	counter9337: LREAL :=  0;
	counter9338: LREAL :=  0;
	counter9339: LREAL :=  0;
	counter9340: LREAL :=  0;
	counter9341: LREAL :=  0;
	counter9342: LREAL :=  0;
	counter9343: LREAL :=  0;
	counter9344: LREAL :=  0;
	counter9345: LREAL :=  0;
	counter9346: LREAL :=  0;
	counter9347: LREAL :=  0;
	counter9348: LREAL :=  0;
	counter9349: LREAL :=  0;
	counter9350: LREAL :=  0;
	counter9351: LREAL :=  0;
	counter9352: LREAL :=  0;
	counter9353: LREAL :=  0;
	counter9354: LREAL :=  0;
	counter9355: LREAL :=  0;
	counter9356: LREAL :=  0;
	counter9357: LREAL :=  0;
	counter9358: LREAL :=  0;
	counter9359: LREAL :=  0;
	counter9360: LREAL :=  0;
	counter9361: LREAL :=  0;
	counter9362: LREAL :=  0;
	counter9363: LREAL :=  0;
	counter9364: LREAL :=  0;
	counter9365: LREAL :=  0;
	counter9366: LREAL :=  0;
	counter9367: LREAL :=  0;
	counter9368: LREAL :=  0;
	counter9369: LREAL :=  0;
	counter9370: LREAL :=  0;
	counter9371: LREAL :=  0;
	counter9372: LREAL :=  0;
	counter9373: LREAL :=  0;
	counter9374: LREAL :=  0;
	counter9375: LREAL :=  0;
	counter9376: LREAL :=  0;
	counter9377: LREAL :=  0;
	counter9378: LREAL :=  0;
	counter9379: LREAL :=  0;
	counter9380: LREAL :=  0;
	counter9381: LREAL :=  0;
	counter9382: LREAL :=  0;
	counter9383: LREAL :=  0;
	counter9384: LREAL :=  0;
	counter9385: LREAL :=  0;
	counter9386: LREAL :=  0;
	counter9387: LREAL :=  0;
	counter9388: LREAL :=  0;
	counter9389: LREAL :=  0;
	counter9390: LREAL :=  0;
	counter9391: LREAL :=  0;
	counter9392: LREAL :=  0;
	counter9393: LREAL :=  0;
	counter9394: LREAL :=  0;
	counter9395: LREAL :=  0;
	counter9396: LREAL :=  0;
	counter9397: LREAL :=  0;
	counter9398: LREAL :=  0;
	counter9399: LREAL :=  0;
	counter9400: LREAL :=  0;
	counter9401: LREAL :=  0;
	counter9402: LREAL :=  0;
	counter9403: LREAL :=  0;
	counter9404: LREAL :=  0;
	counter9405: LREAL :=  0;
	counter9406: LREAL :=  0;
	counter9407: LREAL :=  0;
	counter9408: LREAL :=  0;
	counter9409: LREAL :=  0;
	counter9410: LREAL :=  0;
	counter9411: LREAL :=  0;
	counter9412: LREAL :=  0;
	counter9413: LREAL :=  0;
	counter9414: LREAL :=  0;
	counter9415: LREAL :=  0;
	counter9416: LREAL :=  0;
	counter9417: LREAL :=  0;
	counter9418: LREAL :=  0;
	counter9419: LREAL :=  0;
	counter9420: LREAL :=  0;
	counter9421: LREAL :=  0;
	counter9422: LREAL :=  0;
	counter9423: LREAL :=  0;
	counter9424: LREAL :=  0;
	counter9425: LREAL :=  0;
	counter9426: LREAL :=  0;
	counter9427: LREAL :=  0;
	counter9428: LREAL :=  0;
	counter9429: LREAL :=  0;
	counter9430: LREAL :=  0;
	counter9431: LREAL :=  0;
	counter9432: LREAL :=  0;
	counter9433: LREAL :=  0;
	counter9434: LREAL :=  0;
	counter9435: LREAL :=  0;
	counter9436: LREAL :=  0;
	counter9437: LREAL :=  0;
	counter9438: LREAL :=  0;
	counter9439: LREAL :=  0;
	counter9440: LREAL :=  0;
	counter9441: LREAL :=  0;
	counter9442: LREAL :=  0;
	counter9443: LREAL :=  0;
	counter9444: LREAL :=  0;
	counter9445: LREAL :=  0;
	counter9446: LREAL :=  0;
	counter9447: LREAL :=  0;
	counter9448: LREAL :=  0;
	counter9449: LREAL :=  0;
	counter9450: LREAL :=  0;
	counter9451: LREAL :=  0;
	counter9452: LREAL :=  0;
	counter9453: LREAL :=  0;
	counter9454: LREAL :=  0;
	counter9455: LREAL :=  0;
	counter9456: LREAL :=  0;
	counter9457: LREAL :=  0;
	counter9458: LREAL :=  0;
	counter9459: LREAL :=  0;
	counter9460: LREAL :=  0;
	counter9461: LREAL :=  0;
	counter9462: LREAL :=  0;
	counter9463: LREAL :=  0;
	counter9464: LREAL :=  0;
	counter9465: LREAL :=  0;
	counter9466: LREAL :=  0;
	counter9467: LREAL :=  0;
	counter9468: LREAL :=  0;
	counter9469: LREAL :=  0;
	counter9470: LREAL :=  0;
	counter9471: LREAL :=  0;
	counter9472: LREAL :=  0;
	counter9473: LREAL :=  0;
	counter9474: LREAL :=  0;
	counter9475: LREAL :=  0;
	counter9476: LREAL :=  0;
	counter9477: LREAL :=  0;
	counter9478: LREAL :=  0;
	counter9479: LREAL :=  0;
	counter9480: LREAL :=  0;
	counter9481: LREAL :=  0;
	counter9482: LREAL :=  0;
	counter9483: LREAL :=  0;
	counter9484: LREAL :=  0;
	counter9485: LREAL :=  0;
	counter9486: LREAL :=  0;
	counter9487: LREAL :=  0;
	counter9488: LREAL :=  0;
	counter9489: LREAL :=  0;
	counter9490: LREAL :=  0;
	counter9491: LREAL :=  0;
	counter9492: LREAL :=  0;
	counter9493: LREAL :=  0;
	counter9494: LREAL :=  0;
	counter9495: LREAL :=  0;
	counter9496: LREAL :=  0;
	counter9497: LREAL :=  0;
	counter9498: LREAL :=  0;
	counter9499: LREAL :=  0;
	counter9500: LREAL :=  0;
	counter9501: LREAL :=  0;
	counter9502: LREAL :=  0;
	counter9503: LREAL :=  0;
	counter9504: LREAL :=  0;
	counter9505: LREAL :=  0;
	counter9506: LREAL :=  0;
	counter9507: LREAL :=  0;
	counter9508: LREAL :=  0;
	counter9509: LREAL :=  0;
	counter9510: LREAL :=  0;
	counter9511: LREAL :=  0;
	counter9512: LREAL :=  0;
	counter9513: LREAL :=  0;
	counter9514: LREAL :=  0;
	counter9515: LREAL :=  0;
	counter9516: LREAL :=  0;
	counter9517: LREAL :=  0;
	counter9518: LREAL :=  0;
	counter9519: LREAL :=  0;
	counter9520: LREAL :=  0;
	counter9521: LREAL :=  0;
	counter9522: LREAL :=  0;
	counter9523: LREAL :=  0;
	counter9524: LREAL :=  0;
	counter9525: LREAL :=  0;
	counter9526: LREAL :=  0;
	counter9527: LREAL :=  0;
	counter9528: LREAL :=  0;
	counter9529: LREAL :=  0;
	counter9530: LREAL :=  0;
	counter9531: LREAL :=  0;
	counter9532: LREAL :=  0;
	counter9533: LREAL :=  0;
	counter9534: LREAL :=  0;
	counter9535: LREAL :=  0;
	counter9536: LREAL :=  0;
	counter9537: LREAL :=  0;
	counter9538: LREAL :=  0;
	counter9539: LREAL :=  0;
	counter9540: LREAL :=  0;
	counter9541: LREAL :=  0;
	counter9542: LREAL :=  0;
	counter9543: LREAL :=  0;
	counter9544: LREAL :=  0;
	counter9545: LREAL :=  0;
	counter9546: LREAL :=  0;
	counter9547: LREAL :=  0;
	counter9548: LREAL :=  0;
	counter9549: LREAL :=  0;
	counter9550: LREAL :=  0;
	counter9551: LREAL :=  0;
	counter9552: LREAL :=  0;
	counter9553: LREAL :=  0;
	counter9554: LREAL :=  0;
	counter9555: LREAL :=  0;
	counter9556: LREAL :=  0;
	counter9557: LREAL :=  0;
	counter9558: LREAL :=  0;
	counter9559: LREAL :=  0;
	counter9560: LREAL :=  0;
	counter9561: LREAL :=  0;
	counter9562: LREAL :=  0;
	counter9563: LREAL :=  0;
	counter9564: LREAL :=  0;
	counter9565: LREAL :=  0;
	counter9566: LREAL :=  0;
	counter9567: LREAL :=  0;
	counter9568: LREAL :=  0;
	counter9569: LREAL :=  0;
	counter9570: LREAL :=  0;
	counter9571: LREAL :=  0;
	counter9572: LREAL :=  0;
	counter9573: LREAL :=  0;
	counter9574: LREAL :=  0;
	counter9575: LREAL :=  0;
	counter9576: LREAL :=  0;
	counter9577: LREAL :=  0;
	counter9578: LREAL :=  0;
	counter9579: LREAL :=  0;
	counter9580: LREAL :=  0;
	counter9581: LREAL :=  0;
	counter9582: LREAL :=  0;
	counter9583: LREAL :=  0;
	counter9584: LREAL :=  0;
	counter9585: LREAL :=  0;
	counter9586: LREAL :=  0;
	counter9587: LREAL :=  0;
	counter9588: LREAL :=  0;
	counter9589: LREAL :=  0;
	counter9590: LREAL :=  0;
	counter9591: LREAL :=  0;
	counter9592: LREAL :=  0;
	counter9593: LREAL :=  0;
	counter9594: LREAL :=  0;
	counter9595: LREAL :=  0;
	counter9596: LREAL :=  0;
	counter9597: LREAL :=  0;
	counter9598: LREAL :=  0;
	counter9599: LREAL :=  0;
	counter9600: LREAL :=  0;
	counter9601: LREAL :=  0;
	counter9602: LREAL :=  0;
	counter9603: LREAL :=  0;
	counter9604: LREAL :=  0;
	counter9605: LREAL :=  0;
	counter9606: LREAL :=  0;
	counter9607: LREAL :=  0;
	counter9608: LREAL :=  0;
	counter9609: LREAL :=  0;
	counter9610: LREAL :=  0;
	counter9611: LREAL :=  0;
	counter9612: LREAL :=  0;
	counter9613: LREAL :=  0;
	counter9614: LREAL :=  0;
	counter9615: LREAL :=  0;
	counter9616: LREAL :=  0;
	counter9617: LREAL :=  0;
	counter9618: LREAL :=  0;
	counter9619: LREAL :=  0;
	counter9620: LREAL :=  0;
	counter9621: LREAL :=  0;
	counter9622: LREAL :=  0;
	counter9623: LREAL :=  0;
	counter9624: LREAL :=  0;
	counter9625: LREAL :=  0;
	counter9626: LREAL :=  0;
	counter9627: LREAL :=  0;
	counter9628: LREAL :=  0;
	counter9629: LREAL :=  0;
	counter9630: LREAL :=  0;
	counter9631: LREAL :=  0;
	counter9632: LREAL :=  0;
	counter9633: LREAL :=  0;
	counter9634: LREAL :=  0;
	counter9635: LREAL :=  0;
	counter9636: LREAL :=  0;
	counter9637: LREAL :=  0;
	counter9638: LREAL :=  0;
	counter9639: LREAL :=  0;
	counter9640: LREAL :=  0;
	counter9641: LREAL :=  0;
	counter9642: LREAL :=  0;
	counter9643: LREAL :=  0;
	counter9644: LREAL :=  0;
	counter9645: LREAL :=  0;
	counter9646: LREAL :=  0;
	counter9647: LREAL :=  0;
	counter9648: LREAL :=  0;
	counter9649: LREAL :=  0;
	counter9650: LREAL :=  0;
	counter9651: LREAL :=  0;
	counter9652: LREAL :=  0;
	counter9653: LREAL :=  0;
	counter9654: LREAL :=  0;
	counter9655: LREAL :=  0;
	counter9656: LREAL :=  0;
	counter9657: LREAL :=  0;
	counter9658: LREAL :=  0;
	counter9659: LREAL :=  0;
	counter9660: LREAL :=  0;
	counter9661: LREAL :=  0;
	counter9662: LREAL :=  0;
	counter9663: LREAL :=  0;
	counter9664: LREAL :=  0;
	counter9665: LREAL :=  0;
	counter9666: LREAL :=  0;
	counter9667: LREAL :=  0;
	counter9668: LREAL :=  0;
	counter9669: LREAL :=  0;
	counter9670: LREAL :=  0;
	counter9671: LREAL :=  0;
	counter9672: LREAL :=  0;
	counter9673: LREAL :=  0;
	counter9674: LREAL :=  0;
	counter9675: LREAL :=  0;
	counter9676: LREAL :=  0;
	counter9677: LREAL :=  0;
	counter9678: LREAL :=  0;
	counter9679: LREAL :=  0;
	counter9680: LREAL :=  0;
	counter9681: LREAL :=  0;
	counter9682: LREAL :=  0;
	counter9683: LREAL :=  0;
	counter9684: LREAL :=  0;
	counter9685: LREAL :=  0;
	counter9686: LREAL :=  0;
	counter9687: LREAL :=  0;
	counter9688: LREAL :=  0;
	counter9689: LREAL :=  0;
	counter9690: LREAL :=  0;
	counter9691: LREAL :=  0;
	counter9692: LREAL :=  0;
	counter9693: LREAL :=  0;
	counter9694: LREAL :=  0;
	counter9695: LREAL :=  0;
	counter9696: LREAL :=  0;
	counter9697: LREAL :=  0;
	counter9698: LREAL :=  0;
	counter9699: LREAL :=  0;
	counter9700: LREAL :=  0;
	counter9701: LREAL :=  0;
	counter9702: LREAL :=  0;
	counter9703: LREAL :=  0;
	counter9704: LREAL :=  0;
	counter9705: LREAL :=  0;
	counter9706: LREAL :=  0;
	counter9707: LREAL :=  0;
	counter9708: LREAL :=  0;
	counter9709: LREAL :=  0;
	counter9710: LREAL :=  0;
	counter9711: LREAL :=  0;
	counter9712: LREAL :=  0;
	counter9713: LREAL :=  0;
	counter9714: LREAL :=  0;
	counter9715: LREAL :=  0;
	counter9716: LREAL :=  0;
	counter9717: LREAL :=  0;
	counter9718: LREAL :=  0;
	counter9719: LREAL :=  0;
	counter9720: LREAL :=  0;
	counter9721: LREAL :=  0;
	counter9722: LREAL :=  0;
	counter9723: LREAL :=  0;
	counter9724: LREAL :=  0;
	counter9725: LREAL :=  0;
	counter9726: LREAL :=  0;
	counter9727: LREAL :=  0;
	counter9728: LREAL :=  0;
	counter9729: LREAL :=  0;
	counter9730: LREAL :=  0;
	counter9731: LREAL :=  0;
	counter9732: LREAL :=  0;
	counter9733: LREAL :=  0;
	counter9734: LREAL :=  0;
	counter9735: LREAL :=  0;
	counter9736: LREAL :=  0;
	counter9737: LREAL :=  0;
	counter9738: LREAL :=  0;
	counter9739: LREAL :=  0;
	counter9740: LREAL :=  0;
	counter9741: LREAL :=  0;
	counter9742: LREAL :=  0;
	counter9743: LREAL :=  0;
	counter9744: LREAL :=  0;
	counter9745: LREAL :=  0;
	counter9746: LREAL :=  0;
	counter9747: LREAL :=  0;
	counter9748: LREAL :=  0;
	counter9749: LREAL :=  0;
	counter9750: LREAL :=  0;
	counter9751: LREAL :=  0;
	counter9752: LREAL :=  0;
	counter9753: LREAL :=  0;
	counter9754: LREAL :=  0;
	counter9755: LREAL :=  0;
	counter9756: LREAL :=  0;
	counter9757: LREAL :=  0;
	counter9758: LREAL :=  0;
	counter9759: LREAL :=  0;
	counter9760: LREAL :=  0;
	counter9761: LREAL :=  0;
	counter9762: LREAL :=  0;
	counter9763: LREAL :=  0;
	counter9764: LREAL :=  0;
	counter9765: LREAL :=  0;
	counter9766: LREAL :=  0;
	counter9767: LREAL :=  0;
	counter9768: LREAL :=  0;
	counter9769: LREAL :=  0;
	counter9770: LREAL :=  0;
	counter9771: LREAL :=  0;
	counter9772: LREAL :=  0;
	counter9773: LREAL :=  0;
	counter9774: LREAL :=  0;
	counter9775: LREAL :=  0;
	counter9776: LREAL :=  0;
	counter9777: LREAL :=  0;
	counter9778: LREAL :=  0;
	counter9779: LREAL :=  0;
	counter9780: LREAL :=  0;
	counter9781: LREAL :=  0;
	counter9782: LREAL :=  0;
	counter9783: LREAL :=  0;
	counter9784: LREAL :=  0;
	counter9785: LREAL :=  0;
	counter9786: LREAL :=  0;
	counter9787: LREAL :=  0;
	counter9788: LREAL :=  0;
	counter9789: LREAL :=  0;
	counter9790: LREAL :=  0;
	counter9791: LREAL :=  0;
	counter9792: LREAL :=  0;
	counter9793: LREAL :=  0;
	counter9794: LREAL :=  0;
	counter9795: LREAL :=  0;
	counter9796: LREAL :=  0;
	counter9797: LREAL :=  0;
	counter9798: LREAL :=  0;
	counter9799: LREAL :=  0;
	counter9800: LREAL :=  0;
	counter9801: LREAL :=  0;
	counter9802: LREAL :=  0;
	counter9803: LREAL :=  0;
	counter9804: LREAL :=  0;
	counter9805: LREAL :=  0;
	counter9806: LREAL :=  0;
	counter9807: LREAL :=  0;
	counter9808: LREAL :=  0;
	counter9809: LREAL :=  0;
	counter9810: LREAL :=  0;
	counter9811: LREAL :=  0;
	counter9812: LREAL :=  0;
	counter9813: LREAL :=  0;
	counter9814: LREAL :=  0;
	counter9815: LREAL :=  0;
	counter9816: LREAL :=  0;
	counter9817: LREAL :=  0;
	counter9818: LREAL :=  0;
	counter9819: LREAL :=  0;
	counter9820: LREAL :=  0;
	counter9821: LREAL :=  0;
	counter9822: LREAL :=  0;
	counter9823: LREAL :=  0;
	counter9824: LREAL :=  0;
	counter9825: LREAL :=  0;
	counter9826: LREAL :=  0;
	counter9827: LREAL :=  0;
	counter9828: LREAL :=  0;
	counter9829: LREAL :=  0;
	counter9830: LREAL :=  0;
	counter9831: LREAL :=  0;
	counter9832: LREAL :=  0;
	counter9833: LREAL :=  0;
	counter9834: LREAL :=  0;
	counter9835: LREAL :=  0;
	counter9836: LREAL :=  0;
	counter9837: LREAL :=  0;
	counter9838: LREAL :=  0;
	counter9839: LREAL :=  0;
	counter9840: LREAL :=  0;
	counter9841: LREAL :=  0;
	counter9842: LREAL :=  0;
	counter9843: LREAL :=  0;
	counter9844: LREAL :=  0;
	counter9845: LREAL :=  0;
	counter9846: LREAL :=  0;
	counter9847: LREAL :=  0;
	counter9848: LREAL :=  0;
	counter9849: LREAL :=  0;
	counter9850: LREAL :=  0;
	counter9851: LREAL :=  0;
	counter9852: LREAL :=  0;
	counter9853: LREAL :=  0;
	counter9854: LREAL :=  0;
	counter9855: LREAL :=  0;
	counter9856: LREAL :=  0;
	counter9857: LREAL :=  0;
	counter9858: LREAL :=  0;
	counter9859: LREAL :=  0;
	counter9860: LREAL :=  0;
	counter9861: LREAL :=  0;
	counter9862: LREAL :=  0;
	counter9863: LREAL :=  0;
	counter9864: LREAL :=  0;
	counter9865: LREAL :=  0;
	counter9866: LREAL :=  0;
	counter9867: LREAL :=  0;
	counter9868: LREAL :=  0;
	counter9869: LREAL :=  0;
	counter9870: LREAL :=  0;
	counter9871: LREAL :=  0;
	counter9872: LREAL :=  0;
	counter9873: LREAL :=  0;
	counter9874: LREAL :=  0;
	counter9875: LREAL :=  0;
	counter9876: LREAL :=  0;
	counter9877: LREAL :=  0;
	counter9878: LREAL :=  0;
	counter9879: LREAL :=  0;
	counter9880: LREAL :=  0;
	counter9881: LREAL :=  0;
	counter9882: LREAL :=  0;
	counter9883: LREAL :=  0;
	counter9884: LREAL :=  0;
	counter9885: LREAL :=  0;
	counter9886: LREAL :=  0;
	counter9887: LREAL :=  0;
	counter9888: LREAL :=  0;
	counter9889: LREAL :=  0;
	counter9890: LREAL :=  0;
	counter9891: LREAL :=  0;
	counter9892: LREAL :=  0;
	counter9893: LREAL :=  0;
	counter9894: LREAL :=  0;
	counter9895: LREAL :=  0;
	counter9896: LREAL :=  0;
	counter9897: LREAL :=  0;
	counter9898: LREAL :=  0;
	counter9899: LREAL :=  0;
	counter9900: LREAL :=  0;
	counter9901: LREAL :=  0;
	counter9902: LREAL :=  0;
	counter9903: LREAL :=  0;
	counter9904: LREAL :=  0;
	counter9905: LREAL :=  0;
	counter9906: LREAL :=  0;
	counter9907: LREAL :=  0;
	counter9908: LREAL :=  0;
	counter9909: LREAL :=  0;
	counter9910: LREAL :=  0;
	counter9911: LREAL :=  0;
	counter9912: LREAL :=  0;
	counter9913: LREAL :=  0;
	counter9914: LREAL :=  0;
	counter9915: LREAL :=  0;
	counter9916: LREAL :=  0;
	counter9917: LREAL :=  0;
	counter9918: LREAL :=  0;
	counter9919: LREAL :=  0;
	counter9920: LREAL :=  0;
	counter9921: LREAL :=  0;
	counter9922: LREAL :=  0;
	counter9923: LREAL :=  0;
	counter9924: LREAL :=  0;
	counter9925: LREAL :=  0;
	counter9926: LREAL :=  0;
	counter9927: LREAL :=  0;
	counter9928: LREAL :=  0;
	counter9929: LREAL :=  0;
	counter9930: LREAL :=  0;
	counter9931: LREAL :=  0;
	counter9932: LREAL :=  0;
	counter9933: LREAL :=  0;
	counter9934: LREAL :=  0;
	counter9935: LREAL :=  0;
	counter9936: LREAL :=  0;
	counter9937: LREAL :=  0;
	counter9938: LREAL :=  0;
	counter9939: LREAL :=  0;
	counter9940: LREAL :=  0;
	counter9941: LREAL :=  0;
	counter9942: LREAL :=  0;
	counter9943: LREAL :=  0;
	counter9944: LREAL :=  0;
	counter9945: LREAL :=  0;
	counter9946: LREAL :=  0;
	counter9947: LREAL :=  0;
	counter9948: LREAL :=  0;
	counter9949: LREAL :=  0;
	counter9950: LREAL :=  0;
	counter9951: LREAL :=  0;
	counter9952: LREAL :=  0;
	counter9953: LREAL :=  0;
	counter9954: LREAL :=  0;
	counter9955: LREAL :=  0;
	counter9956: LREAL :=  0;
	counter9957: LREAL :=  0;
	counter9958: LREAL :=  0;
	counter9959: LREAL :=  0;
	counter9960: LREAL :=  0;
	counter9961: LREAL :=  0;
	counter9962: LREAL :=  0;
	counter9963: LREAL :=  0;
	counter9964: LREAL :=  0;
	counter9965: LREAL :=  0;
	counter9966: LREAL :=  0;
	counter9967: LREAL :=  0;
	counter9968: LREAL :=  0;
	counter9969: LREAL :=  0;
	counter9970: LREAL :=  0;
	counter9971: LREAL :=  0;
	counter9972: LREAL :=  0;
	counter9973: LREAL :=  0;
	counter9974: LREAL :=  0;
	counter9975: LREAL :=  0;
	counter9976: LREAL :=  0;
	counter9977: LREAL :=  0;
	counter9978: LREAL :=  0;
	counter9979: LREAL :=  0;
	counter9980: LREAL :=  0;
	counter9981: LREAL :=  0;
	counter9982: LREAL :=  0;
	counter9983: LREAL :=  0;
	counter9984: LREAL :=  0;
	counter9985: LREAL :=  0;
	counter9986: LREAL :=  0;
	counter9987: LREAL :=  0;
	counter9988: LREAL :=  0;
	counter9989: LREAL :=  0;
	counter9990: LREAL :=  0;
	counter9991: LREAL :=  0;
	counter9992: LREAL :=  0;
	counter9993: LREAL :=  0;
	counter9994: LREAL :=  0;
	counter9995: LREAL :=  0;
	counter9996: LREAL :=  0;
	counter9997: LREAL :=  0;
	counter9998: LREAL :=  0;
	counter9999: LREAL :=  0;
END_VAR

(* stored: Version 1.1.0.1, ProductVersion 3.1.4022.18
   GVL StressTest: Id {a7c39071-9d23-401c-b08e-687ae661c369} *)
